// TIA Portal V15.1 export
// export: Created 2020-06-12T07:35:41.9130859Z, ExportSetting None, DisplayName Totally Integrated Automation Portal, DisplayVersion V15.1, DisplayName TIA Portal Openness, DisplayVersion V15.1, DisplayName STEP 7 Professional, DisplayVersion V15.1, DisplayName STEP 7 Safety, DisplayVersion V15.1, DisplayName WinCC Advanced, DisplayVersion V15.1
DATA_BLOCK "GLOB_VAR"   // DB201
{ S7_Optimized_Access := 'TRUE' }
// stored: MemoryReserve 0
   VAR
      emer_ok : Bool := TRUE;   // Emergency circuit is ok
      cont_volt_ok : Bool := TRUE;   // Mains voltage is on
      pwr_ok { ExternalAccessible := 'False'; ExternalVisible := 'False'; ExternalWritable := 'False'} : Bool := TRUE;   // Power is suplleing
      sd_ok : Bool := TRUE;   // Safety doors are ok (locked)
      ES1GD01_desk_is_act : Bool := FALSE;   // Desk ESMGD01 is active
      ES1GD02_desk_is_act : Bool := FALSE;   // Desk ESMGD02 is active
      ES1GD03_desk_is_act : Bool := FALSE;   // Desk ESMGD03 is active
      ES1GT07_desk_is_act : Bool := FALSE;   // Desk ES1GT07 is active
      ack : Bool := FALSE;   // Acknowledge Button
      horn_on : Bool := FALSE;   // Horn on Signal
      sum_flt : Bool := TRUE;   // Summary fault
   END_VAR
   VAR RETAIN
      emer_mode : Bool := FALSE;   // Emergency mode is active
      emer_elcar_lift_cmd : Bool := FALSE;   // Emergency mode: lift electrode carriage command
   END_VAR
   VAR
      emer_pump_on_cmd : Bool := FALSE;   // Emergency mode: pump ON command
      melt_on : Bool := FALSE;   // Melt is ON
   END_VAR
BEGIN
END_DATA_BLOCK
